// TIA Portal project "modulo222" (V20)

(* hardware
DEVICE "S7-1200 station_1"  S7-1200 Station
   slot 0: "Rack_0"  S7-1200 Rack  Rack  V1.0
   slot 1: "PLC_1"  CPU 1214C DC/DC/DC  6ES7 214-1AG40-0XB0  V4.7
*)

// ===== PLC "PLC_1"  CPU 1214C DC/DC/DC =====

VAR_GLOBAL   // PLC tag table "Default tag table"
   "MOTOR" AT %Q0.0 : Bool;
   "Tag_2" AT %I0.0 : Bool;
   "PARTIDA" AT %M0.0 : Bool;
   "PARADA" AT %M0.1 : Bool;
   "EMERGENCIA" AT %M0.2 : Bool;
END_VAR

ORGANIZATION_BLOCK "Main"   // OB1, LAD, ProgramCycle
TITLE = "Main Program Sweep (Cycle)"
{ S7_Optimized_Access := 'TRUE' }
VERSION : 0.1
   VAR_INPUT
      Initial_Call : Bool;   // Initial call of this OB
      Remanence : Bool;   // =True, if remanent data are available
   END_VAR
BEGIN

REGION Network 2
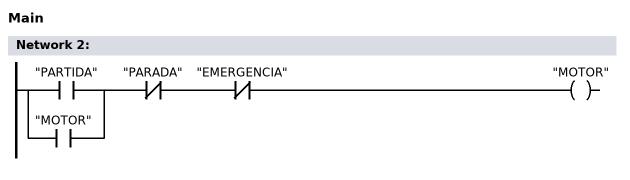
   RUNG wire#powerrail
      Contact( "PARTIDA" )
      wire#w1
      I_Contact( "PARADA" )
      I_Contact( "EMERGENCIA" )
      Coil( "MOTOR" )
   END_RUNG
   RUNG wire#powerrail
      Contact( "MOTOR" )
   END_RUNG wire#w1
   // the same network as SCL:
   "MOTOR" := ("PARTIDA" OR "MOTOR") AND NOT "PARADA" AND NOT "EMERGENCIA";
END_REGION
END_ORGANIZATION_BLOCK